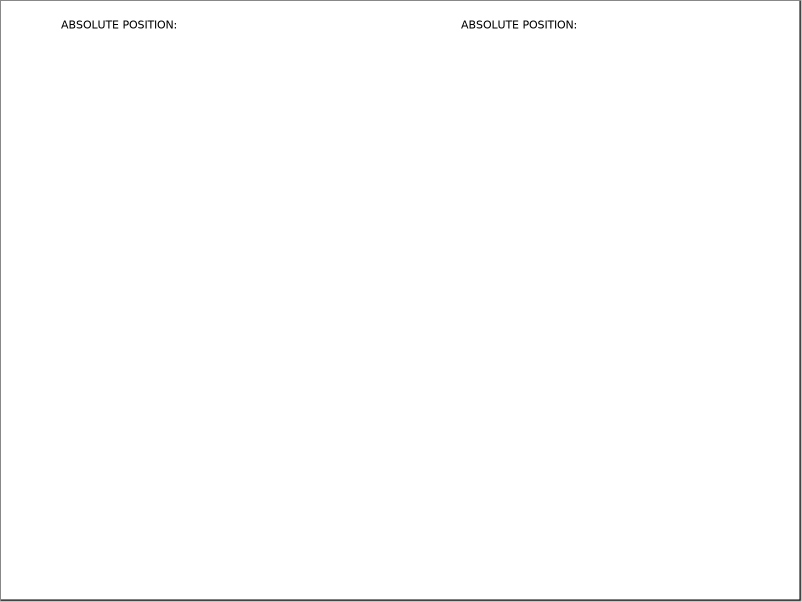
VISUALIZATION F42_Gear_In_Multi_Master  // 802x602
    Rectangle (0,0 800x600)
    Label (10,10 170x30), "ABSOLUTE POSITION:"
    Label (410,10 170x30), "ABSOLUTE POSITION:"
END_VISUALIZATION

(* stored: Version 1.1.0.1, ProductVersion 3.1.4022.7
   Visu F42_Gear_In_Multi_Master: Id {c14a29c8-e859-4ca6-9fb4-e43f1ce8a732} *)
